# EPICS autosave request: measCompApp/Db/USB1208_settings.req
file "measCompBinaryDir_settings.req",      P=$(P), R=Bd1
file "measCompBinaryDir_settings.req",      P=$(P), R=Bd2
file "measCompAnalogInMode_settings.req",   P=$(P), R=AiMode
file "measCompAnalogIn_settings.req",       P=$(P), R=Ai1
file "measCompAnalogIn_settings.req",       P=$(P), R=Ai2
file "measCompAnalogIn_settings.req",       P=$(P), R=Ai3
file "measCompAnalogIn_settings.req",       P=$(P), R=Ai4
file "measCompAnalogOut_settings.req",      P=$(P), R=Ao1
file "measCompAnalogOut_settings.req",      P=$(P), R=Ao2
